// TIA Portal V20 export
DATA_BLOCK "EVTLOG"   // DB950
BEGIN
END_DATA_BLOCK
